VAR_GLOBAL
	g_a_pCtrlInst: ARRAY[0..E_CtrlId.E_CtrlIdMax] OF POINTER TO fb_CtrlBase;
	g_a_pCtrlCIf: ARRAY[0..E_CtrlId.E_CtrlIdMax] OF POINTER TO T_Ctrl_CIf;
	g_fbAlm_Man: FB_Alm_Man;
END_VAR

(* stored: Version 1.1.0.1, ProductVersion 3.1.0.18
   GVL Global: Id {118a3a19-d9ae-43fa-9370-0480fd6e4d03} *)
